TYPE T_TaskNameString : STRING(63); END_TYPE

(* stored: Version 1.1.0.1
   DUT T_TaskNameString: Id {b7424cef-0593-0a3b-0a62-0e929c73ad7d} *)
